(* PLC project robotic_arm, Dassault Systèmes ControlBuild 2024x *)
(* stored: creationDateTime 2023-10-04T11:03:56-01:00 *)

(* This module simulates a single robot arm with rotation calculations *)
FUNCTION_BLOCK motion_control.robotic_arm
  VAR_INPUT
    armOrigin : ARRAY[1..3] OF REAL := [235.0, 2(100.0)];
    overallArmQuatInput : ARRAY[1..4] OF REAL := [1.0, 3(0.0)];
    structRotVector : ARRAY[1..3] OF REAL := [2(0.0), 1.0];
    structRotDeg : REAL := 0.0;
    driveRotVector : ARRAY[1..3] OF REAL := [2(0.0), 1.0];
    driveRotDeg : REAL := 0.0;
    ownRotDeg : REAL := 0.0;
    driveResizeLength : REAL := 0.0;
    functionActive : BOOL := false;
  END_VAR
  VAR_OUTPUT
    armExtrem : ARRAY[1..3] OF REAL := [3(0.0)];
    overallArmRotOutput : ARRAY[1..4] OF REAL := [4(0.0)];
    productId : DINT := -1;
  END_VAR
  VAR
    status_act_prod : DINT := 0;
    m11 : REAL := 1.0;
    m12 : REAL := 0.0;
    m13 : REAL := 0.0;
    m14 : REAL := 0.0;
    m21 : REAL := 0.0;
    m22 : REAL := 1.0;
    m23 : REAL := 0.0;
    m24 : REAL := 0.0;
    m31 : REAL := 0.0;
    m32 : REAL := 0.0;
    m33 : REAL := 1.0;
    m34 : REAL := 0.0;
    m41 : REAL := 0.0;
    m42 : REAL := 0.0;
    m43 : REAL := 0.0;
    m44 : REAL := 1.0;
    armLengthCalc : REAL := 0.0;
    functionActiveLocale : BOOL := false;
    product_id : DINT := -1;
    arm_id : DINT := -1;
    timeToGripParam : REAL := 0.15;
  END_VAR
  VAR CONSTANT
    armLength : REAL := 100.0;
    armWidth : REAL := 5.0;
    armHeight : REAL := 5.0;
    armType : INT := 0;
  END_VAR


ACTION C_source_code:
/* ----------------------------------------------------------------	*/
/* Type : Model of Operative Behaviour					*/
/* Category :  Motion control						*/
/* Author : Dassault Systemes						*/
/* Update date : June 2021							*/
/* ----------------------------------------------------------------	*/
/* This module simulates the behaviour of a robotic arm		*/
/* ----------------------------------------------------------------	*/

arm_id = myself;
productId = product_id; // copy to output for miscelleanous use
product_id = -1;
functionActiveLocale = functionActive;

armLengthCalc = armLength + driveResizeLength;
if (armLengthCalc < 0.0) armLengthCalc = 0.0;

// *** position of current arm relatively to origin ***
double extrem[3];
extrem[0] = armLengthCalc;
extrem[1] = 0;
extrem[2] = 0;

// *** Compute structRotation applying structRotDeg ***
double structAxis[3];
Quaternion structRotation;
structAxis[0] = structRotVector(1); structAxis[1] = structRotVector(2); structAxis[2] = structRotVector(3);
Quaternion_fromAxisAngle(structAxis, structRotDeg*M_PI/180, &structRotation);
Quaternion_normalize(&structRotation, &structRotation);

// *** Compute rotation applying driveRotDeg & ownRotDeg ***
double axis[3];
Quaternion rotation;
axis[0] = driveRotVector(1); axis[1] = driveRotVector(2); axis[2] = driveRotVector(3);
Quaternion_fromAxisAngle(axis, (driveRotDeg + ownRotDeg)*M_PI/180, &rotation);
Quaternion_normalize(&rotation, &rotation);

// *** Get overall quaterniom coming from previous arm ***
Quaternion overall;
overall.w = overallArmQuatInput(1); //w 
overall.v[0] = overallArmQuatInput(2); //cx 
overall.v[1] = overallArmQuatInput(3); //cy 
overall.v[2] = overallArmQuatInput(4); //cz

// *** Add current rotations to get next overall quaternion ***
Quaternion_multiply(&overall, &structRotation, &overall);
Quaternion_multiply(&overall, &rotation, &overall);
overallArmRotOutput(1) = overall.w;
overallArmRotOutput(2) = overall.v[0];
overallArmRotOutput(3) = overall.v[1];
overallArmRotOutput(4) = overall.v[2];

// *** Apply overall rotation to current arm relatively to origin
Quaternion_rotate(&overall, extrem, extrem); 

// *** Shift current arm to previous arm extremity ***
armExtrem(1) = armOrigin(1) + extrem[0];
armExtrem(2) = armOrigin(2) + extrem[1];
armExtrem(3) = armOrigin(3) + extrem[2];

// *** display in ControlBuild coordinate system ***
double eulerAngles[3];
Quaternion_toEulerZYX(&overall , eulerAngles);

if (armLengthCalc == 0.0) armLengthCalc = 0.001;
resizeTo(myself, armLengthCalc, armWidth, armHeight);

rotateTo(myself,0.0 , 0.0 , 0.0, 0.0, 0.0, 0.0);
moveTo(myself, 0.0, -armWidth/2.0, ROT_REFZ-armHeight/2.0);
rotateBy(myself,eulerAngles[0]*180/M_PI ,eulerAngles[1]*180/M_PI ,eulerAngles[2]*180/M_PI, 0.0, 0.0, ROT_REFZ);
moveBy(myself, armOrigin(1), armOrigin(2), armOrigin(3)-ROT_REFZ); 
END_ACTION

ACTION C_header:
#define ROT_REFZ 5000.0// offset of the Z position used for intermediate rotations

#pragma once
#include <stdbool.h>
#include <stdint.h>
#include <stdio.h>
#include <math.h>
#include <stdlib.h>
#include <assert.h>

typedef struct Quaternion {
	double w;	   /**< Scalar part */
	double v[3];	/**< Vector part */
} Quaternion;

void Quaternion_fromAxisAngle(double axis[3], double angle, Quaternion* output);
double Quaternion_norm(Quaternion* q);
void Quaternion_normalize(Quaternion* q, Quaternion* output);
void Quaternion_multiply(Quaternion* q1, Quaternion* q2, Quaternion* output);
void Quaternion_rotate(Quaternion* q, double v[3], double output[3]);

void Quaternion_set(double w, double v1, double v2, double v3, Quaternion* output) {
	output->w = w;
	output->v[0] = v1;
	output->v[1] = v2;
	output->v[2] = v3;
}

void Quaternion_fromAxisAngle(double axis[3], double angle, Quaternion* output) {
	output->w = cos(angle / 2.0);
	double c = sin(angle / 2.0);
	output->v[0] = c * axis[0];
	output->v[1] = c * axis[1];
	output->v[2] = c * axis[2];
}

double Quaternion_norm(Quaternion* q) {
	return sqrt(q->w*q->w + q->v[0]*q->v[0] + q->v[1]*q->v[1] + q->v[2]*q->v[2]);
}

void Quaternion_normalize(Quaternion* q, Quaternion* output) {
	double len = Quaternion_norm(q);
	Quaternion_set(
		q->w / len,
		q->v[0] / len,
		q->v[1] / len,
		q->v[2] / len,
		output);
}

void Quaternion_multiply(Quaternion* q1, Quaternion* q2, Quaternion* output) {
	assert(output != NULL);
	Quaternion result;
	result.w =	q1->w * q2->w - q1->v[0] * q2->v[0] - q1->v[1] * q2->v[1] - q1->v[2] * q2->v[2];
	result.v[0] = q1->v[0] * q2->w + q1->w * q2->v[0] + q1->v[1] * q2->v[2] - q1->v[2] * q2->v[1];
	result.v[1] = q1->w * q2->v[1] - q1->v[0] * q2->v[2] + q1->v[1] * q2->w + q1->v[2] * q2->v[0];
	result.v[2] = q1->w * q2->v[2] + q1->v[0] * q2->v[1] - q1->v[1] * q2->v[0] + q1->v[2] * q2->w   ;

	*output = result;
}

void Quaternion_rotate(Quaternion* q, double v[3], double output[3]) {
	assert(output != NULL);
	double result[3];

	double ww = q->w * q->w;
	double xx = q->v[0] * q->v[0];
	double yy = q->v[1] * q->v[1];
	double zz = q->v[2] * q->v[2];
	double wx = q->w * q->v[0];
	double wy = q->w * q->v[1];
	double wz = q->w * q->v[2];
	double xy = q->v[0] * q->v[1];
	double xz = q->v[0] * q->v[2];
	double yz = q->v[1] * q->v[2];

	result[0] = ww*v[0] + 2*wy*v[2] - 2*wz*v[1] +
				xx*v[0] + 2*xy*v[1] + 2*xz*v[2] -
				zz*v[0] - yy*v[0];
	result[1] = 2*xy*v[0] + yy*v[1] + 2*yz*v[2] +
				2*wz*v[0] - zz*v[1] + ww*v[1] -
				2*wx*v[2] - xx*v[1];
	result[2] = 2*xz*v[0] + 2*yz*v[1] + zz*v[2] -
				2*wy*v[0] - yy*v[2] + 2*wx*v[1] -
				xx*v[2] + ww*v[2];

	output[0] = result[0];
	output[1] = result[1];
	output[2] = result[2];
}

void Quaternion_toEulerZYX(Quaternion* q, double output[3]) {
	assert(output != NULL);

	// Roll (x-axis rotation)
	double sinr_cosp = +2.0 * (q->w * q->v[0] + q->v[1] * q->v[2]);
	double cosr_cosp = +1.0 - 2.0 * (q->v[0] * q->v[0] + q->v[1] * q->v[1]);
	output[0] = atan2(sinr_cosp, cosr_cosp);
	

	// Pitch (y-axis rotation)
	double sinp = +2.0 * (q->w * q->v[1] - q->v[2] * q->v[0]);
	if (fabs(sinp) >= 1)
		output[1] = copysign(M_PI / 2, sinp); // use 90 degrees if out of range
	else
		output[1] = asin(sinp);

	// Yaw (z-axis rotation)
	double siny_cosp = +2.0 * (q->w * q->v[2] + q->v[0] * q->v[1]);
	double cosy_cosp = +1.0 - 2.0 * (q->v[1] * q->v[1] + q->v[2] * q->v[2]);
	output[2] = atan2(siny_cosp, cosy_cosp);
}
END_ACTION
END_FUNCTION_BLOCK
